(* IEC 61131-3 sources: PLC_02/MbTCP/MbTcpS, 3 files *)

(* ---- Types.typ ---- *)
(********************************************************************
 * COPYRIGHT -- Bernecker + Rainer
 ********************************************************************
 * Program: MbApp
 * File: MbApp.typ
 * Author: Bernecker + Rainer
 * Created: October 22, 2009
 ********************************************************************
 * Local data types of program MbApp
 ********************************************************************)

TYPE
	Initial_ParameterType : 	STRUCT
		ModbusStation : STRING[20];
		Coils_startAddress : UINT;
		register_StartAddress : UINT;
		FunctionNum : UDINT;
		RegisterNum : USINT;
		CoilsNum : USINT;
	END_STRUCT;
	ModbusCtrlType : 	STRUCT
		Init_Parameter : Initial_ParameterType;
		Read_Holding_Registers : mbSlWordGet;
		Write_Multiple_Registers : mbSlWordPut;
		Read_Coils : mbSlBoolGet;
		Write_Multiple_Coils : mbSlBoolPut;
		Data : ModbusDataType;
	END_STRUCT;
	ModbusDataType : 	STRUCT
		Coils : ARRAY[0..COILS_NUM_MINUS_1]OF BOOL;
		Register : ARRAY[0..127]OF UINT;
	END_STRUCT;
END_TYPE

(* ---- Main.st ---- *)
PROGRAM _INIT

	ModbusCtrl.Init_Parameter.ModbusStation					:= 'IF2.MODBUSSLAVE_1' ;
	ModbusCtrl.Init_Parameter.register_StartAddress			:= 0 ;
	ModbusCtrl.Init_Parameter.FunctionNum					:= mbMFC_WRITE_MULTIPLE_REGISTERS ;

	fub_status			:= 0;							(* status of function blocks *)
	mb_exception		:= 0;							(* modbus exception *)

END_PROGRAM

PROGRAM _CYCLIC

	(* WORKING STATE MACHINE *)
	CASE (ModbusCtrl.Init_Parameter.FunctionNum) OF

		mbMFC_WRITE_MULTIPLE_REGISTERS: 	// Modbus Function 03

//			memcpy(ADR(ModbusCtrl.Data.Register), ADR(gBAT.ModbusTCP), SIZEOF(gBAT.ModbusTCP) / SIZEOF(gBAT.ModbusTCP.BSA0) );

//			ModbusCtrl.Write_Multiple_Registers(enable := TRUE,
//				startAddress := 16#6000,
//				nrOfItems := SIZEOF(gBAT.ModbusTCP) / SIZEOF(gBAT.ModbusTCP.BSA0),
//				station := ModbusCtrl.Init_Parameter.ModbusStation,
//				data := ModbusCtrl.Data.Register);

			IF (ModbusCtrl.Read_Holding_Registers.status <> ERR_FUB_BUSY) THEN
				fub_status 			:= ModbusCtrl.Write_Multiple_Registers.status;

				check_status 		:= TRUE;			(* flag to check status *)
				instruction_ready 	:= TRUE;			(* flag marks instruction "ready" *)
			ELSE

			END_IF

	END_CASE

	(* ERROR HANDLING *)
	IF (check_status) THEN

		CASE fub_status OF

			ERR_OK:

				gSignalCheck.TCP_Check := TRUE;

			ELSE
   				(* other error handling *)

		END_CASE;

		(* stop checking *)
		check_status := FALSE;
	END_IF

//
//	(* STATE MACHINE CONTROL *)
//	IF (instruction_ready AND fub_status = ERR_OK) THEN
//
//		CASE (instruction) OF
//
//			mbMFC_READ_HOLDING_REGISTERS:
//				instruction 		:= mbMFC_READ_COILS;
//				instruction_ready 	:= FALSE;
//
//			mbMFC_READ_COILS:
//				instruction 		:= mbMFC_READ_HOLDING_REGISTERS;
//				instruction_ready 	:= FALSE;
//
//		END_CASE
//
//	END_IF

END_PROGRAM

(* ---- Variables.var ---- *)
(********************************************************************
 * COPYRIGHT -- Bernecker + Rainer
 ********************************************************************
 * Program: MbApp
 * File: MbApp.var
 * Author: Bernecker + Rainer
 * Created: October 22, 2009
 ********************************************************************
 * Local variables of program MbApp
 ********************************************************************)
VAR
	fub_status : UINT; (*status of function blocks*)
	mb_exception : USINT; (*modbus exception*)
	check_status : BOOL; (*flag to check status*)
	instruction_ready : BOOL; (*flag marks instruction "ready"*)
	ModbusCtrl : ModbusCtrlType;
	HandlingData1 : ARRAY[0..COILS_NUM_MINUS_1] OF BOOL;
	HandlingData2 : ARRAY[0..REGITSTER_NUM_MINUS_1] OF INT;
END_VAR
VAR CONSTANT
	REGITSTER_NUM : USINT := 97;
	COILS_NUM : USINT := 2;
	REGITSTER_NUM_MINUS_1 : USINT := REGITSTER_NUM-1;
	COILS_NUM_MINUS_1 : USINT := COILS_NUM-1;
END_VAR
VAR
	InputWord : UINT;
	InputWord2 : USINT;
	InputWord3 : USINT;
END_VAR
